# EPICS autosave request: iocBoot/ioc2/dbSave/23i_WS_Av_.req
%
% BURT Request File
%
% 23i:WS:Av:  White beam slits, Vertical Aperture
%

file $(DIR)/assy.req ASSY=23i:WS:Av
23i:WS:Av:Invert
file $(DIR)/mtr1.req MTR1=23i:WS:mt
file $(DIR)/mtr1.req MTR1=23i:WS:mb
file $(DIR)/drv1.req DRV1=23i:WS:ZT
file $(DIR)/drv1.req DRV1=23i:WS:ZB
file $(DIR)/axs1.req AXS1=23i:WS:ZC
file $(DIR)/axs1.req AXS1=23i:WS:ZS
